(* LS Electric XG5000 project: PLC_Study *)
(* PLC LSPLC *)
(* module base 0 slot 0: 입력 모듈:XGI-D21A (DC 24V 입력, 8점 (전류소스/싱크입력)) *)
(* module base 0 slot 1: 출력 모듈:XGQ-RY1A (릴레이 출력, 8점 (2A용, 단독 COM.)) *)
(* module base 0 slot 2: 출력 모듈:XGQ-RY1A (릴레이 출력, 8점 (2A용, 단독 COM.)) *)

(* Comments on direct variables
%QX0.1.0	출력
%QX0.1.2	출력
%IX0.0.3	스위치
*)

PROGRAM NewProgram (* task: 스캔 프로그램 *)

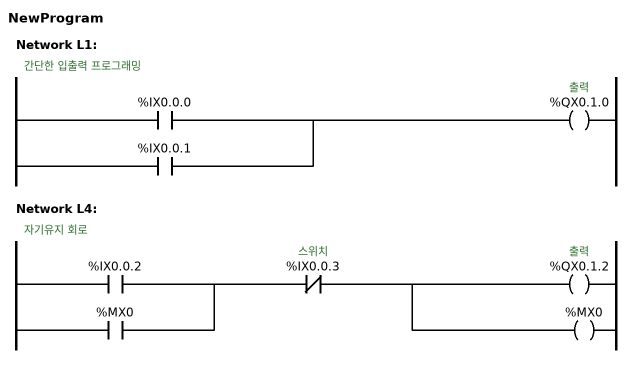
(* 간단한 입출력 프로그래밍 *)
(* Rung L1 *)
%QX0.1.0 := %IX0.0.0 OR %IX0.0.1;
(* 자기유지 회로 *)
(* Rung L4 *)
%QX0.1.2 := (%IX0.0.2 OR %MX0) AND NOT %IX0.0.3;
%MX0 := (%IX0.0.2 OR %MX0) AND NOT %IX0.0.3;
END_PROGRAM

PROGRAM 양음변환검출코일 (* task: 스캔 프로그램 *)
VAR
    삼번스위치 AT %IX0.0.3 : BOOL;
    양변환검출코일 AT %QX0.1.0 : BOOL;
    음변환검출코일 AT %QX0.1.2 : BOOL;
    이번LED AT %QX0.1.3 : BOOL;
    이번스위치 AT %IX0.0.2 : BOOL;
    일번LED AT %QX0.1.1 : BOOL;
    일번스위치 AT %IX0.0.1 : BOOL;
END_VAR
VAR
    _e1 : R_TRIG;
    _e2 : F_TRIG;
END_VAR

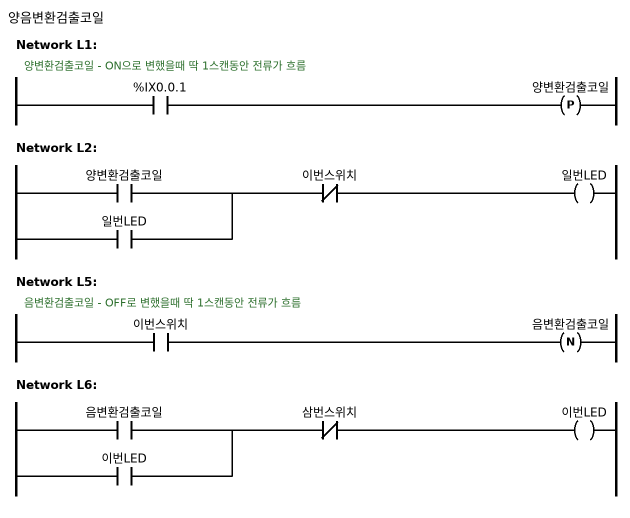
(* 양변환검출코일 - ON으로 변했을때 딱 1스캔동안 전류가 흐름 *)
(* Rung L1 *)
_e1(CLK := %IX0.0.1);
양변환검출코일 := _e1.Q;
(* Rung L2 *)
일번LED := (양변환검출코일 OR 일번LED) AND NOT 이번스위치;
(* 음변환검출코일 - OFF로 변했을때 딱 1스캔동안 전류가 흐름 *)
(* Rung L5 *)
_e2(CLK := 이번스위치);
음변환검출코일 := _e2.Q;
(* Rung L6 *)
이번LED := (음변환검출코일 OR 이번LED) AND NOT 삼번스위치;
END_PROGRAM